(* PLC project LadderFidelityFixture, greenforge-labs codescribe-fixture 1 *)
(* stored: creationDateTime 2020-01-01T00:00:00 *)

PROGRAM LD_FIDELITY
  VAR
    xGo : BOOL;
    xStart : BOOL;
    xManual : BOOL;
    xDone : BOOL;
    iCount : INT;
    ctr : CTU;
    xPress : BOOL;
    xStop : BOOL;
    xRun : BOOL;
    xCool : BOOL;
    tmr2 : TON;
  END_VAR

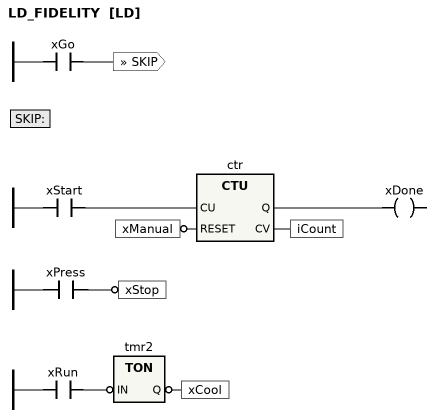
(* LD diagram, written out as Structured Text *)
IF xGo THEN JMP SKIP; END_IF;
SKIP:
ctr(CU := xStart, RESET := NOT xManual, CV => iCount);
xDone := ctr.Q;
xStop := NOT xPress;
tmr2(IN := NOT xRun, Q => xCool);
END_PROGRAM
